// TIA Portal V17 export
// export: Created 2023-06-23T18:33:41.7486641Z, ExportSetting WithDefaults, DisplayName Totally Integrated Automation Portal, DisplayVersion V17, DisplayName TIA Portal Openness, DisplayVersion V17, DisplayName TIA Portal Version Control Interface, DisplayVersion V17, DisplayName STEP 7 Professional, DisplayVersion V17, DisplayName STEP 7 Safety, DisplayVersion V17, DisplayName WinCC Advanced / Unified PC, DisplayVersion V17
VAR_GLOBAL   // PLC tag table "31_BAT-1"
   "iBAT-1" AT %I16.0 : Bool;
   "oBAT-1" AT %Q13.3 : Bool;
END_VAR
